INTERFACE I_Restorable EXTENDS __SYSTEM.IQueryInterface

METHOD Restore : I_Restorable
VAR_INPUT
END_VAR
END_METHOD

END_INTERFACE

(* stored: Version 1.1.0.1, ProductVersion 3.1.4024.12
   Itf I_Restorable: Id {013c2610-d02c-42c6-86e8-03b3b8c8717d}
   Method Restore: Id {3e98e5e0-5ef8-4687-98c2-cba9e3a31fe8} *)
